{attribute addProperty BoxType "EL3011-0000-0016"}
{attribute addProperty Id "AI_StandardAT %I*AI_Standard_B51B79FC8110.1250WcStateAT %I*WcState_F855686C1620InfoDataAT %I*InfoData_BC63D37F80100"}
{attribute addProperty CRC "368140935"}
{attribute addProperty SizeInBites "177"}
{attribute addProperty SizeInBytes "22.125"}
TYPE EL3011_4607B8C0 :
STRUCT
	{attribute addProperty Name "AI_Standard"}
	AI_Standard : AI_Standard_B51B79FC;
	{attribute addProperty Name "WcState"}
	WcState : WcState_F855686C;
	{attribute addProperty Name "InfoData"}
	InfoData : InfoData_BC63D37F;
END_STRUCT
END_TYPE

(* stored: Version 1.2.0.0, ProductVersion 3.1.4024.9
   DUT EL3011_4607B8C0: Id {13f3420d-e858-4f7e-8692-35897413a18d} *)
